(*

short summary
=================
This data type contains just a REAL value and it's string representation.

.. <legal notes>

legal notes
=================
| SPDX-FileCopyrightText: © 2022 ekvip automation GmbH <info@ekvip.de>
| SPDX-License-Identifier: Apache-2.0
| For details check: Apache-2.0_

.. _Apache-2.0: https://www.apache.org/licenses/LICENSE-2.0

.. </legal notes>

type members
======================

*)

TYPE RealTestParameter :
STRUCT
	(* just the value to test *)
	value		:REAL;
	(* string representation of ``value`` *)
	asString	:Tc2_System.T_MaxString;
END_STRUCT
END_TYPE

(* stored: Version 1.1.0.1, ProductVersion 3.1.4026.11
   DUT RealTestParameter: Id {f3f14a58-20c3-4955-afd1-7a96f174f64b} *)
